PROGRAM BasketTotalizer
VAR

END_VAR

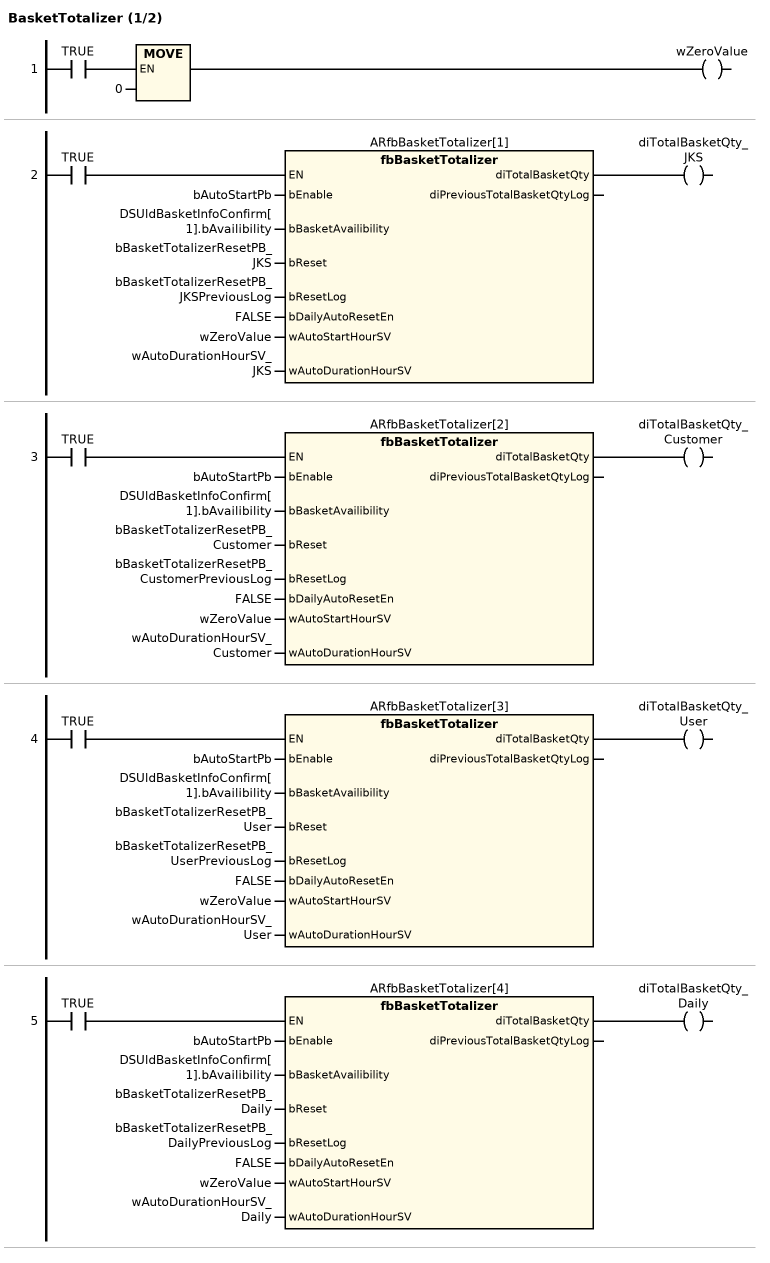
// NETWORK 1
wZeroValue := 0;

// NETWORK 2
ARfbBasketTotalizer[1](
    bEnable := bAutoStartPb,
    bBasketAvailibility := DSUldBasketInfoConfirm[1].bAvailibility,
    bReset := bBasketTotalizerResetPB_JKS,
    bResetLog := bBasketTotalizerResetPB_JKSPreviousLog,
    bDailyAutoResetEn := FALSE,
    wAutoStartHourSV := wZeroValue,
    wAutoDurationHourSV := wAutoDurationHourSV_JKS); // fbBasketTotalizer
diTotalBasketQty_JKS := ARfbBasketTotalizer[1].diTotalBasketQty;

// NETWORK 3
ARfbBasketTotalizer[2](
    bEnable := bAutoStartPb,
    bBasketAvailibility := DSUldBasketInfoConfirm[1].bAvailibility,
    bReset := bBasketTotalizerResetPB_Customer,
    bResetLog := bBasketTotalizerResetPB_CustomerPreviousLog,
    bDailyAutoResetEn := FALSE,
    wAutoStartHourSV := wZeroValue,
    wAutoDurationHourSV := wAutoDurationHourSV_Customer); // fbBasketTotalizer
diTotalBasketQty_Customer := ARfbBasketTotalizer[2].diTotalBasketQty;

// NETWORK 4
ARfbBasketTotalizer[3](
    bEnable := bAutoStartPb,
    bBasketAvailibility := DSUldBasketInfoConfirm[1].bAvailibility,
    bReset := bBasketTotalizerResetPB_User,
    bResetLog := bBasketTotalizerResetPB_UserPreviousLog,
    bDailyAutoResetEn := FALSE,
    wAutoStartHourSV := wZeroValue,
    wAutoDurationHourSV := wAutoDurationHourSV_User); // fbBasketTotalizer
diTotalBasketQty_User := ARfbBasketTotalizer[3].diTotalBasketQty;

// NETWORK 5
ARfbBasketTotalizer[4](
    bEnable := bAutoStartPb,
    bBasketAvailibility := DSUldBasketInfoConfirm[1].bAvailibility,
    bReset := bBasketTotalizerResetPB_Daily,
    bResetLog := bBasketTotalizerResetPB_DailyPreviousLog,
    bDailyAutoResetEn := FALSE,
    wAutoStartHourSV := wZeroValue,
    wAutoDurationHourSV := wAutoDurationHourSV_Daily); // fbBasketTotalizer
diTotalBasketQty_Daily := ARfbBasketTotalizer[4].diTotalBasketQty;

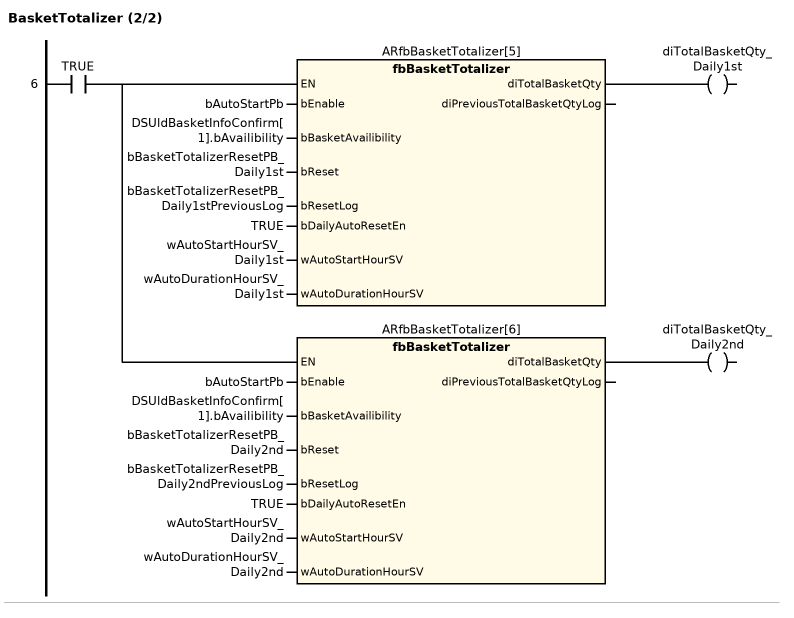
// NETWORK 6
ARfbBasketTotalizer[5](
    bEnable := bAutoStartPb,
    bBasketAvailibility := DSUldBasketInfoConfirm[1].bAvailibility,
    bReset := bBasketTotalizerResetPB_Daily1st,
    bResetLog := bBasketTotalizerResetPB_Daily1stPreviousLog,
    bDailyAutoResetEn := TRUE,
    wAutoStartHourSV := wAutoStartHourSV_Daily1st,
    wAutoDurationHourSV := wAutoDurationHourSV_Daily1st); // fbBasketTotalizer
diTotalBasketQty_Daily1st := ARfbBasketTotalizer[5].diTotalBasketQty;
ARfbBasketTotalizer[6](
    bEnable := bAutoStartPb,
    bBasketAvailibility := DSUldBasketInfoConfirm[1].bAvailibility,
    bReset := bBasketTotalizerResetPB_Daily2nd,
    bResetLog := bBasketTotalizerResetPB_Daily2ndPreviousLog,
    bDailyAutoResetEn := TRUE,
    wAutoStartHourSV := wAutoStartHourSV_Daily2nd,
    wAutoDurationHourSV := wAutoDurationHourSV_Daily2nd); // fbBasketTotalizer
diTotalBasketQty_Daily2nd := ARfbBasketTotalizer[6].diTotalBasketQty;

END_PROGRAM

(* stored: Version 1.1.0.1, ProductVersion 3.1.4024.12
   POU BasketTotalizer: Id {d062475c-bba7-400b-8bd7-bbf89051b8ef}, SpecialFunc None *)
